INTERFACE I_Alarm

PROPERTY AlarmNumber : UINT
GET
END_GET
SET
END_SET
END_PROPERTY

PROPERTY Description : String
GET
END_GET
SET
END_SET
END_PROPERTY

METHOD Get : BOOL
VAR_INPUT
END_VAR
VAR_OUTPUT

END_VAR
END_METHOD

METHOD Reset : BOOL
VAR_INPUT
END_VAR
END_METHOD

METHOD Set : BOOL
VAR
END_VAR
VAR_INPUT
	bIn	:	BOOL;
END_VAR
END_METHOD

PROPERTY TimeOfOccur : TIMESTRUCT
GET
END_GET
END_PROPERTY

END_INTERFACE

(* stored: Version 1.1.0.1, ProductVersion 3.1.4024.12
   Itf I_Alarm: Id {44119e1c-5e4e-4538-bd9b-92dbca0e41e4}
   Property AlarmNumber: Id {93e32961-c723-4eba-acfc-789f4f11fcfe}
   Get Get: Id {450326d5-e627-416e-9af2-58e4419f9fbb}
   Set Set: Id {f1a51338-04b6-48c6-863f-af5e96f31833}
   Property Description: Id {b387e12b-f56b-420a-9bc1-39aaf6ff001b}
   Get Get: Id {c3b34a70-d556-49b0-8c1e-9c498f607d00}
   Set Set: Id {f598d613-8a01-4bdd-b514-96aec54ec3c0}
   Method Get: Id {e0c3f08b-6fd0-4bb5-b0ca-719ca49a193c}
   Method Reset: Id {0ae1005c-0204-452e-b861-401b524b3cbf}
   Method Set: Id {6a93a594-3088-41f7-9da4-29944c40752a}
   Property TimeOfOccur: Id {36f6e22d-3214-4cec-893f-a095cfb32990}
   Get Get: Id {22e2ce27-af3c-4886-b33f-4787f3576304} *)
